% RSLogix 500 project LVD190506v3_Top.RSS, saved by version 11.00.00.00 %
PROJECT "LINCEBOT"    % processor: MicroLogix 1400 %

PROGRAM FILES
  LAD 2 "MAIN"  63 rungs  % Main Program Routine %
  LAD 8 "LOOP TIME"  6 rungs
  LAD 12 "ENABLES"  4 rungs
  LAD 14 "SPEED OUT"  3 rungs
  LAD 16 "TOTALCOUNT"  4 rungs
  LAD 19 "TESTTRIG5"  4 rungs
  LAD 20 "TESTTRIG6"  4 rungs
  LAD 21 "TESTTRIG7"  4 rungs
  LAD 22 "TESTTRIG8"  4 rungs
  LAD 24 "SKIPPED"  5 rungs
  LAD 26 "TEST TIME"  11 rungs
  LAD 70 "ALIGNFAILS"  4 rungs  % normal %
  LAD 90 "HSC TOP"  5 rungs
  LAD 100 "1 MS STI"  23 rungs  % high speed %
  LAD 103 "SPEED TOP"  8 rungs  % high speed %
  LAD 105 "P TOP"  7 rungs  % high speed %
  LAD 111 "SHIFT TOP"  15 rungs
  LAD 131 "READXFER"  3 rungs
  LAD 140 "TOP_OPTIC"  8 rungs
  LAD 141 "TOPOP_VERT"  5 rungs
  LAD 142 "TOPOP_REAL"  10 rungs
  LAD 143 "TOPOP_TEST"  13 rungs
  LAD 144 "TOP_OP_OK"  6 rungs
  LAD 150 "TOP_OPTIC"  6 rungs
  LAD 151 "TOPOP_VERT"  9 rungs
  LAD 152 "TOPOP_REAL"  11 rungs
  LAD 153 "TOPOP_TEST"  19 rungs
  LAD 154 "TOP_OP_OK"  6 rungs
  LAD 155 "OP RNG TST"  5 rungs
  LAD 190 "INS5"  21 rungs
  LAD 191 "INS5RESULT"  7 rungs
  LAD 192 "INS5PASS"  4 rungs
  LAD 193 "INS5FAIL"  3 rungs
  LAD 194 "INS5ACQ"  8 rungs
  LAD 195 "Q5TIMETEST"  5 rungs
  LAD 196 "INS5TRIG"  5 rungs
  LAD 197 "FIFO5SET"  9 rungs
  LAD 198 "FIFO5GET"  8 rungs
  LAD 199 "INSDATA5"  3 rungs
  LAD 200 "TESTFAULT5"  9 rungs
  LAD 201 "INS5FIX1"  6 rungs
  LAD 202 "INS5FIX2"  3 rungs
  LAD 204 "INS6"  21 rungs
  LAD 205 "INS6RESULT"  7 rungs
  LAD 206 "INS6PASS"  4 rungs
  LAD 207 "INS6FAIL"  3 rungs
  LAD 208 "INS6ACQ"  8 rungs
  LAD 209 "Q6TIMETEST"  5 rungs
  LAD 210 "INS6TRIG"  5 rungs
  LAD 211 "FIFO6SET"  9 rungs
  LAD 212 "FIFO6GET"  8 rungs
  LAD 213 "INSDATA6"  3 rungs
  LAD 214 "TESTFAULT6"  9 rungs
  LAD 215 "INS6FIX1"  6 rungs
  LAD 216 "INS6FIX2"  3 rungs
  LAD 218 "INS7"  21 rungs
  LAD 219 "INS7RESULT"  7 rungs
  LAD 220 "INS7PASS"  4 rungs
  LAD 221 "INS7FAIL"  3 rungs
  LAD 222 "INS7ACQ"  8 rungs
  LAD 223 "Q7TIMETEST"  5 rungs
  LAD 224 "INS7TRIG"  5 rungs
  LAD 225 "FIFO7SET"  9 rungs
  LAD 226 "FIFO7GET"  8 rungs
  LAD 227 "INSDATA7"  3 rungs
  LAD 228 "TESTFAULT7"  9 rungs
  LAD 229 "INS7FIX1"  6 rungs
  LAD 230 "INS7FIX2"  3 rungs
  LAD 232 "INS8"  21 rungs
  LAD 233 "INS8RESULT"  7 rungs
  LAD 234 "INS8PASS"  4 rungs
  LAD 235 "INS8FAIL"  3 rungs
  LAD 236 "INS8ACQ"  8 rungs
  LAD 237 "Q8TIMETEST"  5 rungs
  LAD 238 "INS8TRIG"  5 rungs
  LAD 239 "FIFO8SET"  9 rungs
  LAD 240 "FIFO8GET"  8 rungs
  LAD 241 "INSDATA8"  3 rungs
  LAD 242 "TESTFAULT8"  9 rungs
  LAD 243 "INS8FIX1"  6 rungs
  LAD 244 "INS8FIX2"  3 rungs
  LAD 249 "PASS BLOW"  25 rungs
  LAD 250 "RECERK"  10 rungs
  LAD 251 "RECERK SET"  5 rungs
  LAD 252 "RATE1"  9 rungs
  LAD 253 "RATE2"  6 rungs
  LAD 254 "RESET RATE"  6 rungs
  LAD 255 "UNUSED"  19 rungs
  LAD 149, 189, 203, 217, 231, 245: only END

DATA FILES
  O0 OUTPUT  6 elements
  I1 INPUT  8 elements
  S2 STATUS  66 elements
  B3 BINARY  64 elements
  T4 TIMER  40 elements
  C5 COUNTER  1 elements
  R6 CONTROL  20 elements
  N7 INTEGER  200 elements
  F8 FLOAT  100 elements
  B9   1 elements
  B10   1 elements
  B11   1 elements
  B12 HMI_BINARY  22 elements  % general use with hmi to avoid additional reads %
  L13  COUNTS  256 elements
  F14 HMI_FLOATS  100 elements
  N15 HMI_INTS  100 elements
  L16 HMI_LONGS  100 elements
  B17 #1 GOOD  192 elements
  B18 #2 GOOD  192 elements
  L19 I5TIMEFIFO  50 elements
  L20 I5POSFIFO  50 elements
  L21 I6TIMEFIFO  50 elements
  L22 I6POSFIFO  50 elements
  L23 I7TIMEFIFO  50 elements
  L24 I7POSFIFO  50 elements
  L25 I8TIMEFIFO  50 elements
  L26 I8POSFIFO  50 elements
  L27 RATE FIFO  50 elements
  L42 COMS  52 elements
  RI43 RI1  11 elements
  MG44 MSG1  11 elements
  B181 BLANK  256 elements  % used to wipe bs files %
  F182   50 elements
  L183   50 elements
  N184   50 elements
  B185   50 elements
  N186   50 elements
  L187   50 elements
  F188   50 elements
  B189   50 elements
  L190   50 elements
  B191   10 elements
  L192 SPD OFFSET  50 elements
  F193 SPD OFFSET  50 elements
  B194 TOP GOOD  192 elements
  B195 TOP NG  192 elements
  B196 CTRL BITS  50 elements
  N197 CTRL INTS  50 elements
  B198 TRK BITS  50 elements
  L199 TRK LONG  50 elements
  N200 TRK INTS  50 elements
  L201 INS LONG  50 elements
  B202 INS BITS  50 elements
  N203 INS INTS  50 elements
  L204 CTRL LONG  50 elements
  F205 CTRL FLTS  50 elements

LADDER 2 "MAIN"    % Main Program Routine %
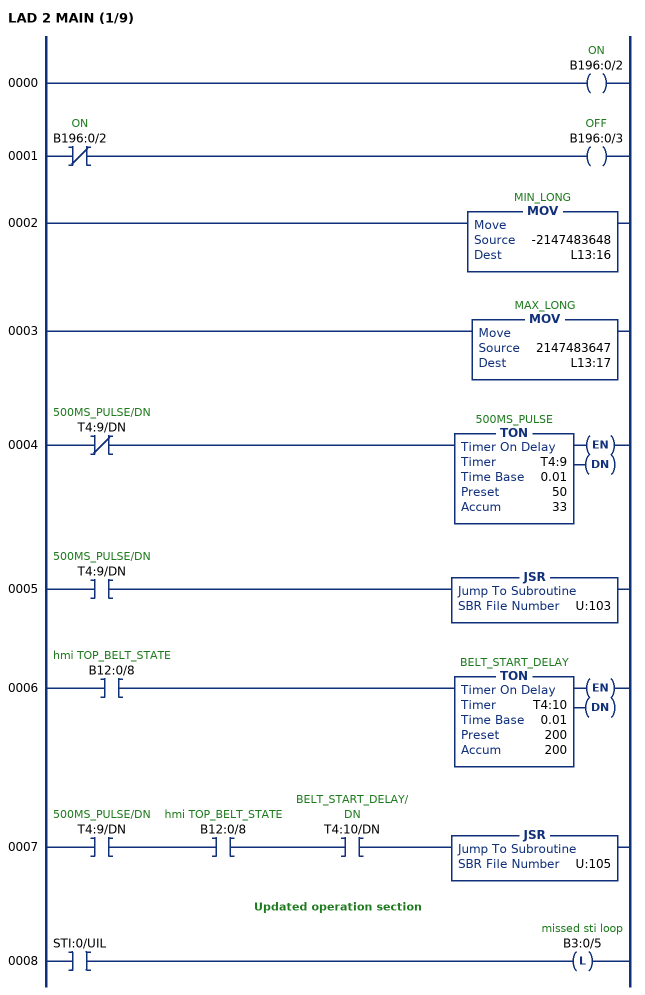
% Rung: 0 %
SOR OTE B196:0/2 EOR
%   B196:0/2  ON %
% Rung: 1 %
SOR XIO B196:0/2 OTE B196:0/3 EOR
%   B196:0/2  ON %
%   B196:0/3  OFF %
% Rung: 2 %
SOR MOV -2147483648 L13:16 EOR
%   L13:16  MIN_LONG %
% Rung: 3 %
SOR MOV 2147483647 L13:17 EOR
%   L13:17  MAX_LONG %
% Rung: 4 %
SOR XIO T4:9/DN TON T4:9 0.01 50 33 EOR
%   T4:9  500MS_PULSE %
% Rung: 5 %
SOR XIC T4:9/DN JSR U:103 EOR
%   T4:9  500MS_PULSE %
% Rung: 6 %
SOR XIC B12:0/8 TON T4:10 0.01 200 200 EOR
%   B12:0/8  TOP_BELT_STATE  "hmi" %
%   T4:10  BELT_START_DELAY %
% Rung: 7 %
SOR XIC T4:9/DN XIC B12:0/8 XIC T4:10/DN JSR U:105 EOR
%   T4:9  500MS_PULSE %
%   B12:0/8  TOP_BELT_STATE  "hmi" %
%   T4:10  BELT_START_DELAY %
% Rung: 8 %
% TITLE: Updated operation section %
SOR XIC STI:0/UIL OTL B3:0/5 EOR
%   B3:0/5  "missed sti loop" %

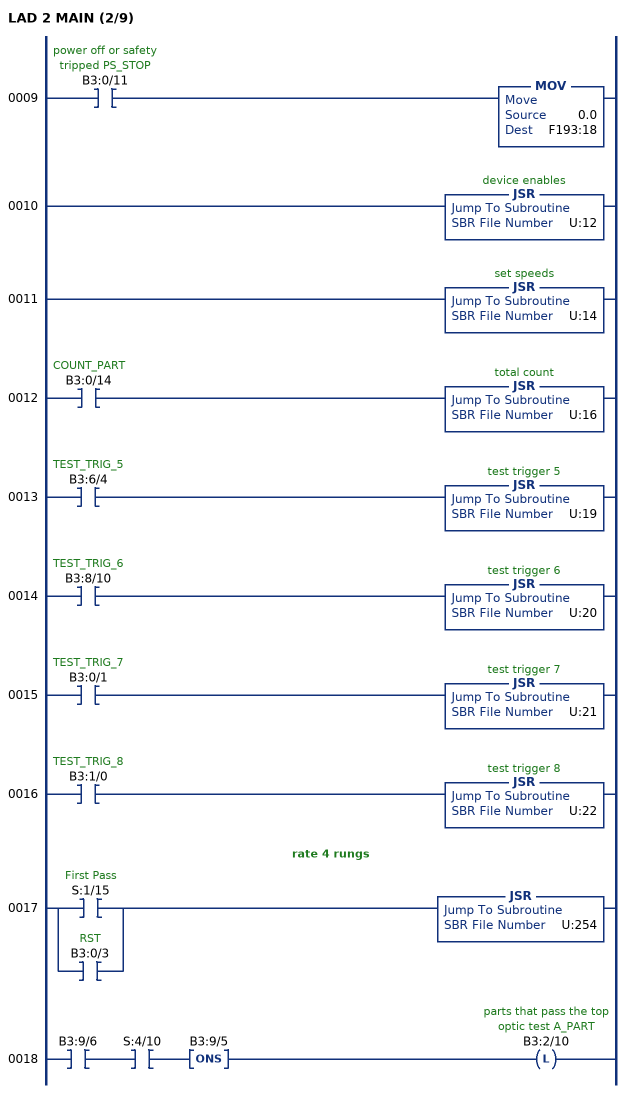
% Rung: 9 %
SOR XIC B3:0/11 MOV 0.0 F193:18 EOR
%   B3:0/11  PS_STOP  "power off or safety tripped" %
% Rung: 10 %
SOR JSR U:12 EOR
%   U:12  "device enables" %
% Rung: 11 %
SOR JSR U:14 EOR
%   U:14  "set speeds" %
% Rung: 12 %
SOR XIC B3:0/14 JSR U:16 EOR
%   B3:0/14  COUNT_PART %
%   U:16  "total count" %
% Rung: 13 %
SOR XIC B3:6/4 JSR U:19 EOR
%   B3:6/4  TEST_TRIG_5 %
%   U:19  "test trigger 5" %
% Rung: 14 %
SOR XIC B3:8/10 JSR U:20 EOR
%   B3:8/10  TEST_TRIG_6 %
%   U:20  "test trigger 6" %
% Rung: 15 %
SOR XIC B3:0/1 JSR U:21 EOR
%   B3:0/1  TEST_TRIG_7 %
%   U:21  "test trigger 7" %
% Rung: 16 %
SOR XIC B3:1/0 JSR U:22 EOR
%   B3:1/0  TEST_TRIG_8 %
%   U:22  "test trigger 8" %
% Rung: 17 %
% TITLE: rate 4 rungs %
SOR BST XIC S:1/15 NXB XIC B3:0/3 BND JSR U:254 EOR
%   S:1/15  "First Pass" %
%   B3:0/3  RST %
% Rung: 18 %
SOR XIC B3:9/6 XIC S:4/10 ONS B3:9/5 OTL B3:2/10 EOR
%   B3:2/10  A_PART  "parts that pass the top optic test" %

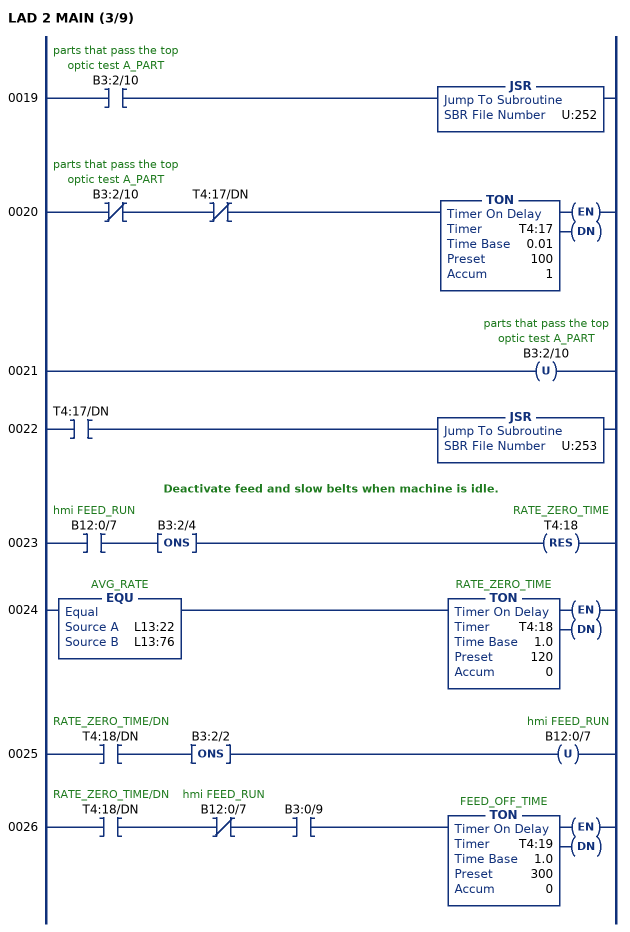
% Rung: 19 %
SOR XIC B3:2/10 JSR U:252 EOR
%   B3:2/10  A_PART  "parts that pass the top optic test" %
% Rung: 20 %
SOR XIO B3:2/10 XIO T4:17/DN TON T4:17 0.01 100 1 EOR
%   B3:2/10  A_PART  "parts that pass the top optic test" %
% Rung: 21 %
SOR OTU B3:2/10 EOR
%   B3:2/10  A_PART  "parts that pass the top optic test" %
% Rung: 22 %
SOR XIC T4:17/DN JSR U:253 EOR
% Rung: 23 %
% TITLE: Deactivate feed and slow belts when machine is idle. %
SOR XIC B12:0/7 ONS B3:2/4 RES T4:18 EOR
%   B12:0/7  FEED_RUN  "hmi" %
%   T4:18  RATE_ZERO_TIME %
% Rung: 24 %
SOR EQU L13:22 L13:76 TON T4:18 1.0 120 0 EOR
%   L13:22  AVG_RATE %
%   L13:76  PPM_AVG %
%   T4:18  RATE_ZERO_TIME %
% Rung: 25 %
SOR XIC T4:18/DN ONS B3:2/2 OTU B12:0/7 EOR
%   T4:18  RATE_ZERO_TIME %
%   B12:0/7  FEED_RUN  "hmi" %
% Rung: 26 %
SOR XIC T4:18/DN XIO B12:0/7 XIC B3:0/9 TON T4:19 1.0 300 0 EOR
%   T4:18  RATE_ZERO_TIME %
%   B12:0/7  FEED_RUN  "hmi" %
%   T4:19  FEED_OFF_TIME %

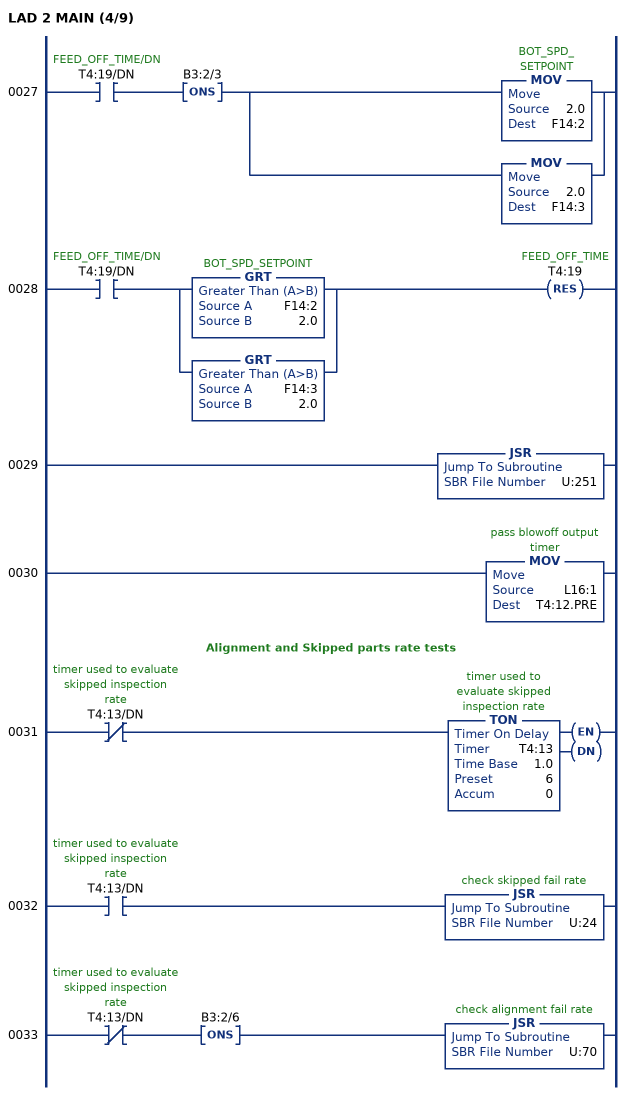
% Rung: 27 %
SOR XIC T4:19/DN ONS B3:2/3 BST MOV 2.0 F14:2 NXB MOV 2.0 F14:3 BND EOR
%   T4:19  FEED_OFF_TIME %
%   F14:2  BOT_SPD_SETPOINT %
% Rung: 28 %
SOR XIC T4:19/DN BST GRT F14:2 2.0 NXB GRT F14:3 2.0 BND RES T4:19 EOR
%   T4:19  FEED_OFF_TIME %
%   F14:2  BOT_SPD_SETPOINT %
% Rung: 29 %
SOR JSR U:251 EOR
% Rung: 30 %
SOR MOV L16:1 T4:12.PRE EOR
%   L16:1  BLOW_TIME %
%   T4:12  "pass blowoff output timer" %
% Rung: 31 %
% TITLE: Alignment and Skipped parts rate tests %
SOR XIO T4:13/DN TON T4:13 1.0 6 0 EOR
%   T4:13  "timer used to evaluate skipped inspection rate" %
% Rung: 32 %
SOR XIC T4:13/DN JSR U:24 EOR
%   T4:13  "timer used to evaluate skipped inspection rate" %
%   U:24  "check skipped fail rate" %
% Rung: 33 %
SOR XIO T4:13/DN ONS B3:2/6 JSR U:70 EOR
%   T4:13  "timer used to evaluate skipped inspection rate" %
%   U:70  "check alignment fail rate" %

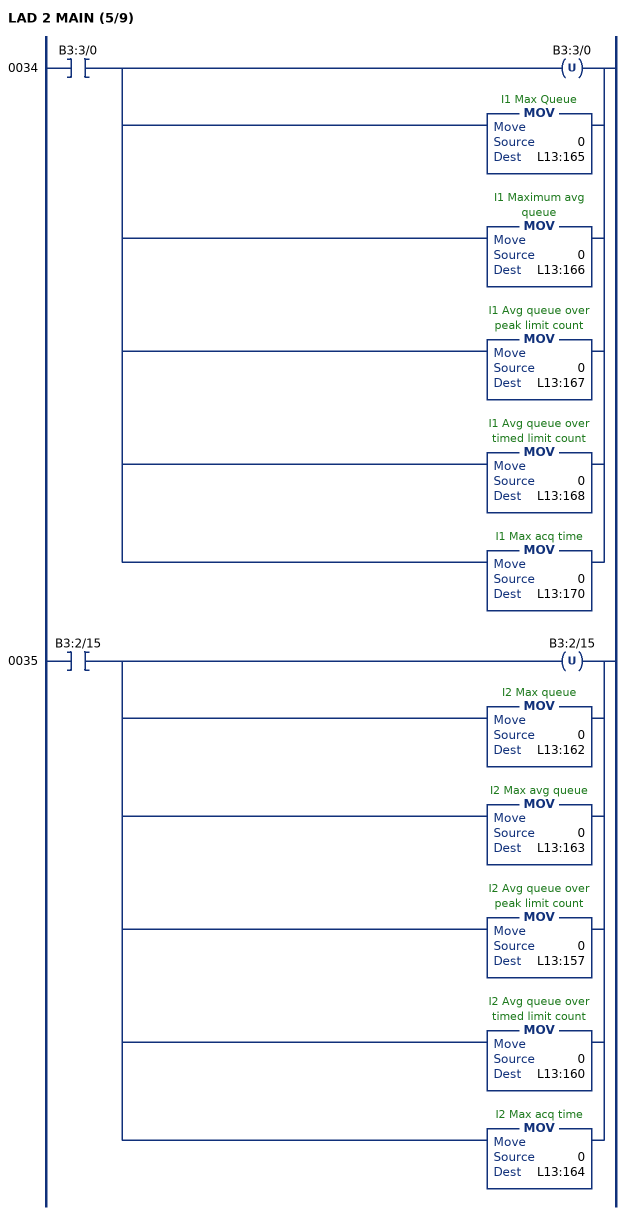
% Rung: 34 %
SOR XIC B3:3/0 BST OTU B3:3/0 NXB MOV 0 L13:165 NXB MOV 0 L13:166 NXB MOV 0 L13:167 NXB MOV 0 L13:168 NXB MOV 0 L13:170 BND EOR
%   L13:165  "I1 Max Queue" %
%   L13:166  "I1 Maximum avg queue" %
%   L13:167  "I1 Avg queue over peak limit count" %
%   L13:168  "I1 Avg queue over timed limit count" %
%   L13:170  "I1 Max acq time" %
% Rung: 35 %
SOR XIC B3:2/15 BST OTU B3:2/15 NXB MOV 0 L13:162 NXB MOV 0 L13:163 NXB MOV 0 L13:157 NXB MOV 0 L13:160 NXB MOV 0 L13:164 BND EOR
%   L13:162  "I2 Max queue" %
%   L13:163  "I2 Max avg queue" %
%   L13:157  "I2 Avg queue over peak limit count" %
%   L13:160  "I2 Avg queue over timed limit count" %
%   L13:164  "I2 Max acq time" %

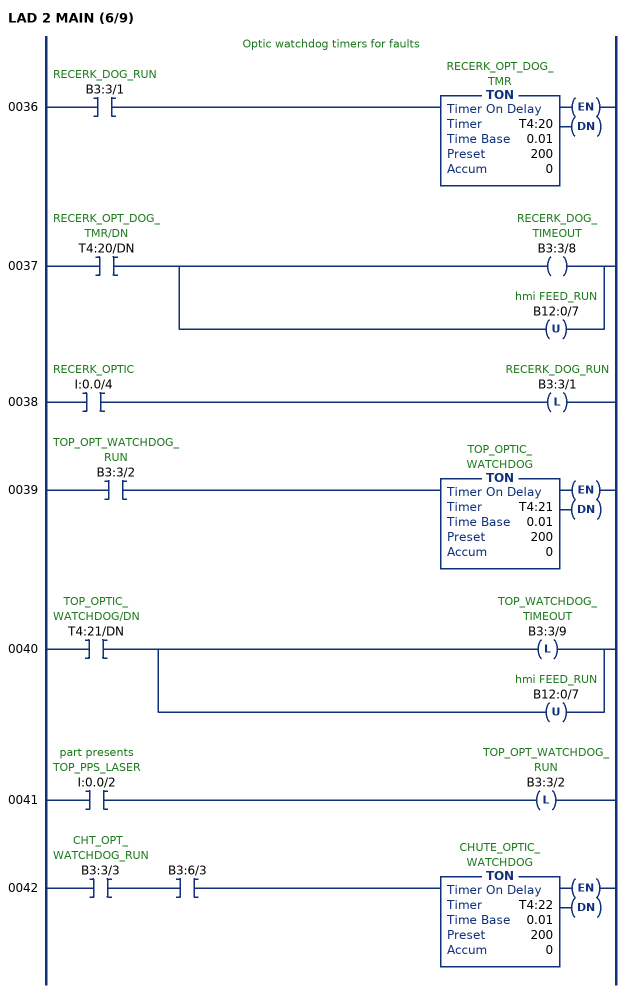
% Rung: 36 %
% Optic watchdog timers for faults %
SOR XIC B3:3/1 TON T4:20 0.01 200 0 EOR
%   B3:3/1  RECERK_DOG_RUN %
%   T4:20  RECERK_OPT_DOG_TMR %
% Rung: 37 %
SOR XIC T4:20/DN BST OTE B3:3/8 NXB OTU B12:0/7 BND EOR
%   T4:20  RECERK_OPT_DOG_TMR %
%   B3:3/8  RECERK_DOG_TIMEOUT %
%   B12:0/7  FEED_RUN  "hmi" %
% Rung: 38 %
SOR XIC I:0.0/4 OTL B3:3/1 EOR
%   I:0.0/4  RECERK_OPTIC %
%   B3:3/1  RECERK_DOG_RUN %
% Rung: 39 %
SOR XIC B3:3/2 TON T4:21 0.01 200 0 EOR
%   B3:3/2  TOP_OPT_WATCHDOG_RUN %
%   T4:21  TOP_OPTIC_WATCHDOG %
% Rung: 40 %
SOR XIC T4:21/DN BST OTL B3:3/9 NXB OTU B12:0/7 BND EOR
%   T4:21  TOP_OPTIC_WATCHDOG %
%   B3:3/9  TOP_WATCHDOG_TIMEOUT %
%   B12:0/7  FEED_RUN  "hmi" %
% Rung: 41 %
SOR XIC I:0.0/2 OTL B3:3/2 EOR
%   I:0.0/2  TOP_PPS_LASER  "part presents" %
%   B3:3/2  TOP_OPT_WATCHDOG_RUN %
% Rung: 42 %
SOR XIC B3:3/3 XIC B3:6/3 TON T4:22 0.01 200 0 EOR
%   B3:3/3  CHT_OPT_WATCHDOG_RUN %
%   T4:22  CHUTE_OPTIC_WATCHDOG %

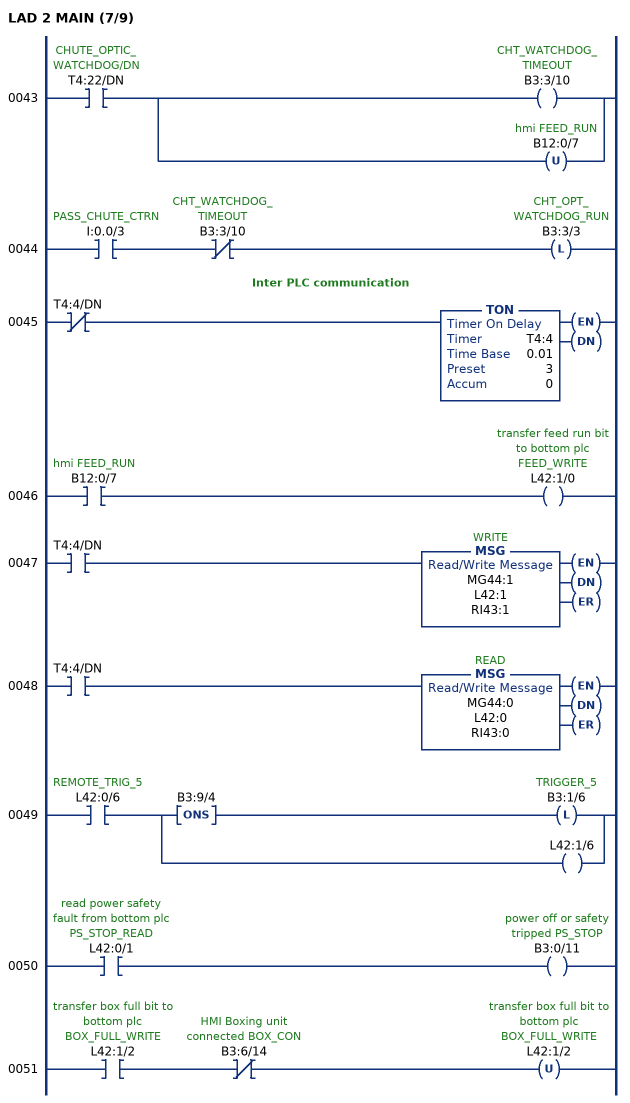
% Rung: 43 %
SOR XIC T4:22/DN BST OTE B3:3/10 NXB OTU B12:0/7 BND EOR
%   T4:22  CHUTE_OPTIC_WATCHDOG %
%   B3:3/10  CHT_WATCHDOG_TIMEOUT %
%   B12:0/7  FEED_RUN  "hmi" %
% Rung: 44 %
SOR XIC I:0.0/3 XIO B3:3/10 OTL B3:3/3 EOR
%   I:0.0/3  PASS_CHUTE_CTRN %
%   B3:3/10  CHT_WATCHDOG_TIMEOUT %
%   B3:3/3  CHT_OPT_WATCHDOG_RUN %
% Rung: 45 %
% TITLE: Inter PLC communication %
SOR XIO T4:4/DN TON T4:4 0.01 3 0 EOR
% Rung: 46 %
SOR XIC B12:0/7 OTE L42:1/0 EOR
%   B12:0/7  FEED_RUN  "hmi" %
%   L42:1/0  FEED_WRITE  "transfer feed run bit to bottom plc" %
% Rung: 47 %
SOR XIC T4:4/DN MSG MG44:1 L42:1 RI43:1 EOR
%   MSG set-up: 500CPU Write | 33 | 1 | L42:0 | L42:1 | 0 | 0 | 0 | 192.168.222.100:0 | 0 | 0 | 192.168.222.100 | RI43:1 %
%   MG44:1  WRITE %
%   L42:1  WRITE_BITS %
% Rung: 48 %
SOR XIC T4:4/DN MSG MG44:0 L42:0 RI43:0 EOR
%   MSG set-up: 500CPU Read | 33 | 1 | L42:1 | L42:0 | 0 | 0 | 0 | 192.168.222.100:0 | 0 | 0 | 192.168.222.100 | RI43:0 %
%   MG44:0  READ %
%   L42:0  READ_BITS %
% Rung: 49 %
SOR XIC L42:0/6 BST ONS B3:9/4 OTL B3:1/6 NXB OTE L42:1/6 BND EOR
%   L42:0/6  REMOTE_TRIG_5 %
%   B3:1/6  TRIGGER_5 %
% Rung: 50 %
SOR XIC L42:0/1 OTE B3:0/11 EOR
%   L42:0/1  PS_STOP_READ  "read power safety fault from bottom plc" %
%   B3:0/11  PS_STOP  "power off or safety tripped" %
% Rung: 51 %
SOR XIC L42:1/2 XIO B3:6/14 OTU L42:1/2 EOR
%   L42:1/2  BOX_FULL_WRITE  "transfer box full bit to bottom plc" %
%   B3:6/14  BOX_CON  "HMI Boxing unit connected" %

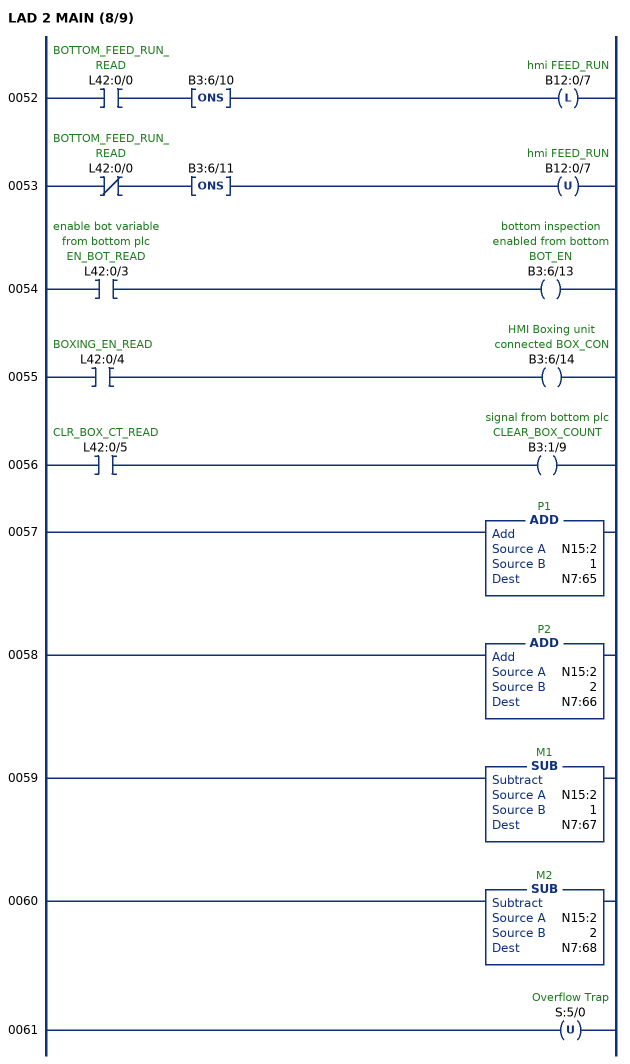
% Rung: 52 %
SOR XIC L42:0/0 ONS B3:6/10 OTL B12:0/7 EOR
%   L42:0/0  BOTTOM_FEED_RUN_READ %
%   B12:0/7  FEED_RUN  "hmi" %
% Rung: 53 %
SOR XIO L42:0/0 ONS B3:6/11 OTU B12:0/7 EOR
%   L42:0/0  BOTTOM_FEED_RUN_READ %
%   B12:0/7  FEED_RUN  "hmi" %
% Rung: 54 %
SOR XIC L42:0/3 OTE B3:6/13 EOR
%   L42:0/3  EN_BOT_READ  "enable bot variable from bottom plc" %
%   B3:6/13  BOT_EN  "bottom inspection enabled from bottom" %
% Rung: 55 %
SOR XIC L42:0/4 OTE B3:6/14 EOR
%   L42:0/4  BOXING_EN_READ %
%   B3:6/14  BOX_CON  "HMI Boxing unit connected" %
% Rung: 56 %
SOR XIC L42:0/5 OTE B3:1/9 EOR
%   L42:0/5  CLR_BOX_CT_READ %
%   B3:1/9  CLEAR_BOX_COUNT  "signal from bottom plc" %
% Rung: 57 %
SOR ADD N15:2 1 N7:65 EOR
%   N15:2  BLOW_PT %
%   N7:65  P1 %
% Rung: 58 %
SOR ADD N15:2 2 N7:66 EOR
%   N15:2  BLOW_PT %
%   N7:66  P2 %
% Rung: 59 %
SOR SUB N15:2 1 N7:67 EOR
%   N15:2  BLOW_PT %
%   N7:67  M1 %
% Rung: 60 %
SOR SUB N15:2 2 N7:68 EOR
%   N15:2  BLOW_PT %
%   N7:68  M2 %
% Rung: 61 %
SOR OTU S:5/0 EOR
%   S:5/0  "Overflow Trap" %

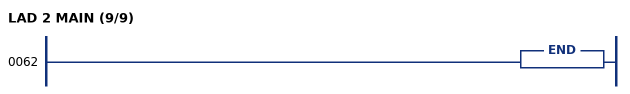
% Rung: 62 %
SOR END EOR

LADDER 8 "LOOP TIME"
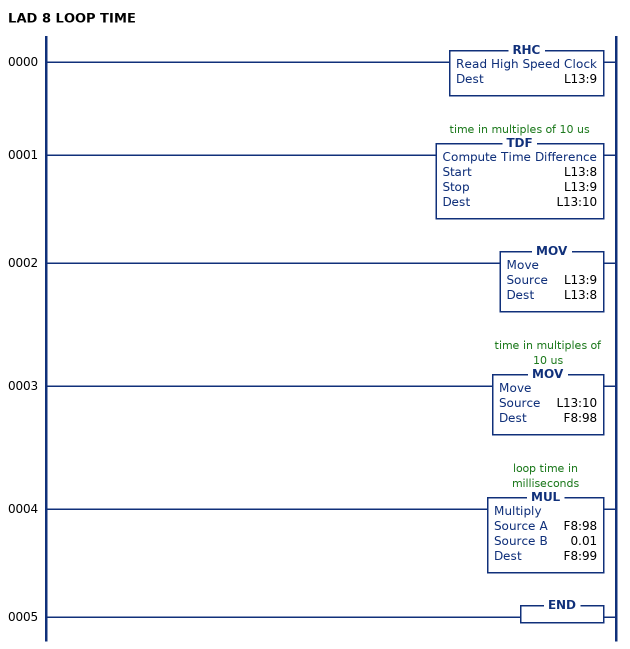
% Rung: 0 %
SOR RHC L13:9 EOR
% Rung: 1 %
SOR TDF L13:8 L13:9 L13:10 EOR
%   L13:10  "time in multiples of 10 us" %
% Rung: 2 %
SOR MOV L13:9 L13:8 EOR
% Rung: 3 %
SOR MOV L13:10 F8:98 EOR
%   L13:10  "time in multiples of 10 us" %
%   F8:98  "time in multiples of 10 us" %
% Rung: 4 %
SOR MUL F8:98 0.01 F8:99 EOR
%   F8:98  "time in multiples of 10 us" %
%   F8:99  "loop time in milliseconds" %
% Rung: 5 %
SOR END EOR

LADDER 12 "ENABLES"
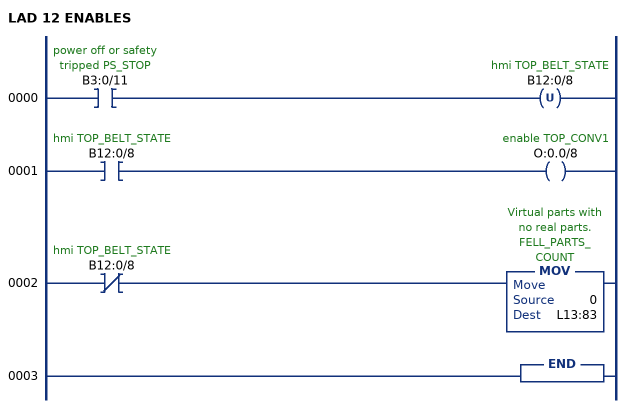
% Rung: 0 %
SOR XIC B3:0/11 OTU B12:0/8 EOR
%   B3:0/11  PS_STOP  "power off or safety tripped" %
%   B12:0/8  TOP_BELT_STATE  "hmi" %
% Rung: 1 %
SOR XIC B12:0/8 OTE O:0.0/8 EOR
%   B12:0/8  TOP_BELT_STATE  "hmi" %
%   O:0.0/8  TOP_CONV1  "enable" %
% Rung: 2 %
SOR XIO B12:0/8 MOV 0 L13:83 EOR
%   B12:0/8  TOP_BELT_STATE  "hmi" %
%   L13:83  FELL_PARTS_COUNT  "Virtual parts with no real parts." %
% Rung: 3 %
SOR END EOR

LADDER 14 "SPEED OUT"
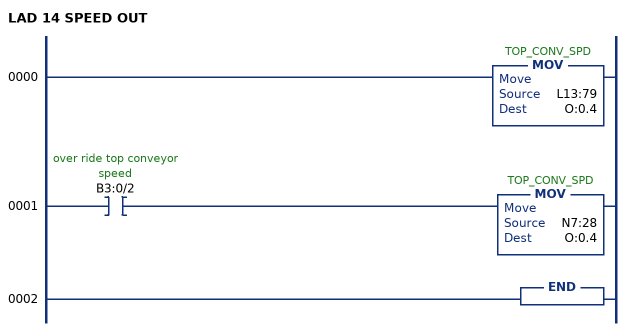
% Rung: 0 %
SOR MOV L13:79 O:0.4 EOR
%   L13:79  SCALED_TOP_VALUE %
%   O:0.4  TOP_CONV_SPD %
% Rung: 1 %
SOR XIC B3:0/2 MOV N7:28 O:0.4 EOR
%   B3:0/2  "over ride top conveyor speed" %
%   O:0.4  TOP_CONV_SPD %
% Rung: 2 %
SOR END EOR

LADDER 16 "TOTALCOUNT"
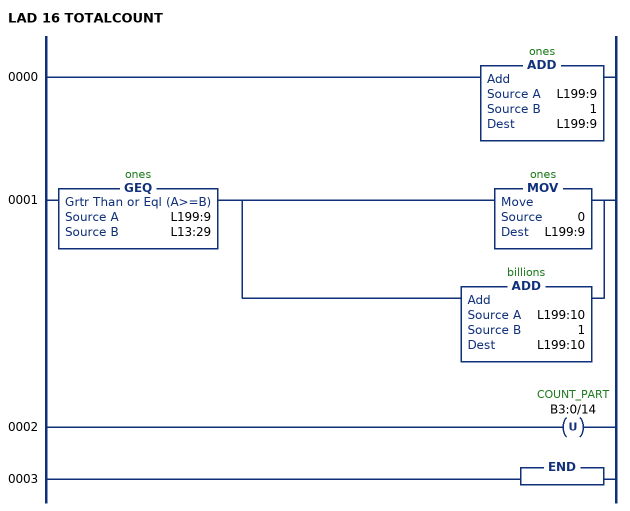
% Rung: 0 %
SOR ADD L199:9 1 L199:9 EOR
%   L199:9  "ones" %
% Rung: 1 %
SOR GEQ L199:9 L13:29 BST MOV 0 L199:9 NXB ADD L199:10 1 L199:10 BND EOR
%   L199:9  "ones" %
%   L13:29  "maximum of the longest acquire time allowed if maximum acquire time fault is enabled" %
%   L199:10  "billions" %
% Rung: 2 %
SOR OTU B3:0/14 EOR
%   B3:0/14  COUNT_PART %
% Rung: 3 %
SOR END EOR

LADDER 19 "TESTTRIG5"
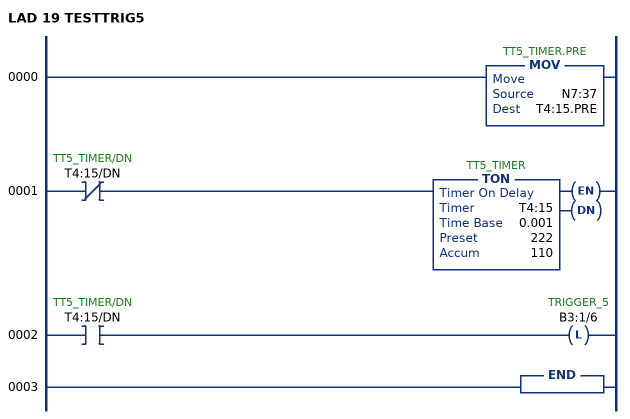
% Rung: 0 %
SOR MOV N7:37 T4:15.PRE EOR
%   T4:15  TT5_TIMER %
% Rung: 1 %
SOR XIO T4:15/DN TON T4:15 0.001 222 110 EOR
%   T4:15  TT5_TIMER %
% Rung: 2 %
SOR XIC T4:15/DN OTL B3:1/6 EOR
%   T4:15  TT5_TIMER %
%   B3:1/6  TRIGGER_5 %
% Rung: 3 %
SOR END EOR

LADDER 20 "TESTTRIG6"
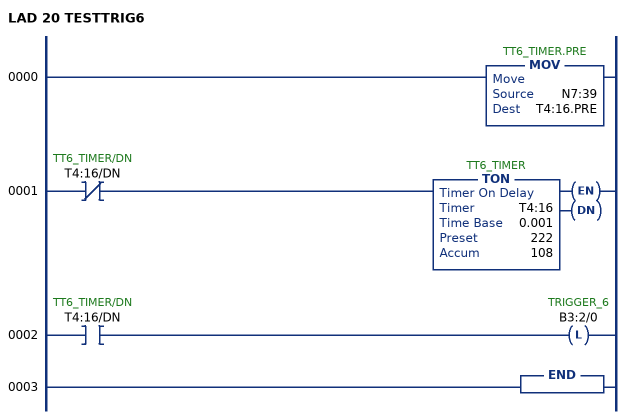
% Rung: 0 %
SOR MOV N7:39 T4:16.PRE EOR
%   T4:16  TT6_TIMER %
% Rung: 1 %
SOR XIO T4:16/DN TON T4:16 0.001 222 108 EOR
%   T4:16  TT6_TIMER %
% Rung: 2 %
SOR XIC T4:16/DN OTL B3:2/0 EOR
%   T4:16  TT6_TIMER %
%   B3:2/0  TRIGGER_6 %
% Rung: 3 %
SOR END EOR

LADDER 21 "TESTTRIG7"
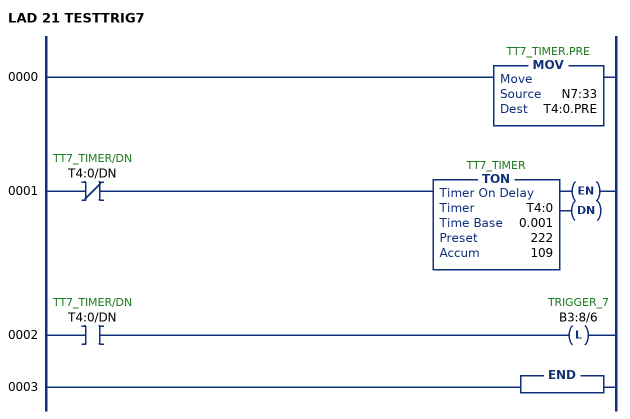
% Rung: 0 %
SOR MOV N7:33 T4:0.PRE EOR
%   T4:0  TT7_TIMER %
% Rung: 1 %
SOR XIO T4:0/DN TON T4:0 0.001 222 109 EOR
%   T4:0  TT7_TIMER %
% Rung: 2 %
SOR XIC T4:0/DN OTL B3:8/6 EOR
%   T4:0  TT7_TIMER %
%   B3:8/6  TRIGGER_7 %
% Rung: 3 %
SOR END EOR

LADDER 22 "TESTTRIG8"
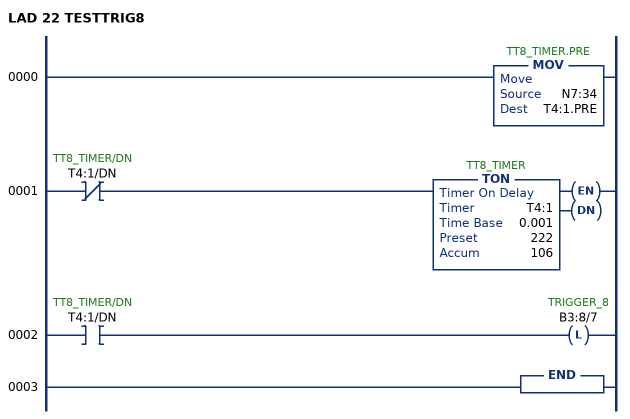
% Rung: 0 %
SOR MOV N7:34 T4:1.PRE EOR
%   T4:1  TT8_TIMER %
% Rung: 1 %
SOR XIO T4:1/DN TON T4:1 0.001 222 106 EOR
%   T4:1  TT8_TIMER %
% Rung: 2 %
SOR XIC T4:1/DN OTL B3:8/7 EOR
%   T4:1  TT8_TIMER %
%   B3:8/7  TRIGGER_8 %
% Rung: 3 %
SOR END EOR

LADDER 24 "SKIPPED"
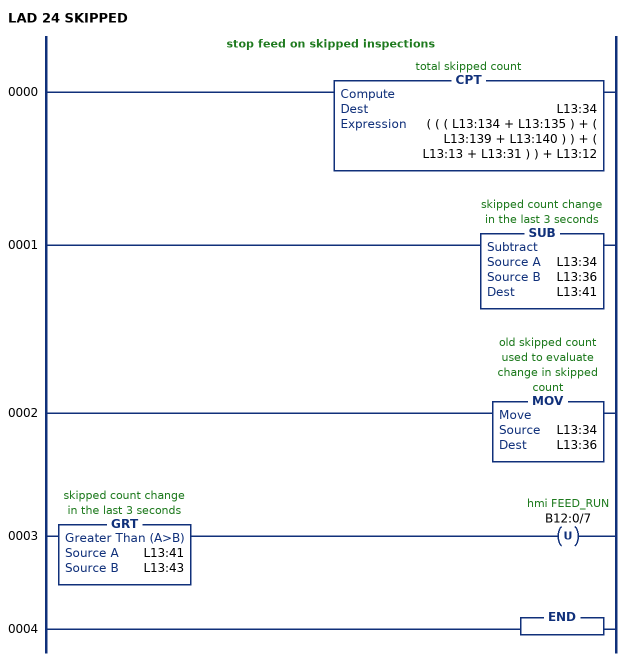
% Rung: 0 %
% TITLE: stop feed on skipped inspections %
SOR CPT L13:34 " ( ( ( L13:134 + L13:135 ) + ( L13:139 + L13:140 ) ) + ( L13:13 + L13:31 ) ) + L13:12 " EOR
%   L13:34  "total skipped count" %
%   L13:134  "too wide bottom" %
%   L13:135  "too close bottom" %
%   L13:139  "too close top count" %
%   L13:140  "too wide top count" %
%   L13:13  SKIP1  "skipped 1 count" %
%   L13:31  SKIP5  "skipped 5 count" %
%   L13:12  SKIP6  "skipped 6 count" %
% Rung: 1 %
SOR SUB L13:34 L13:36 L13:41 EOR
%   L13:34  "total skipped count" %
%   L13:36  "old skipped count used to evaluate change in skipped count" %
%   L13:41  "skipped count change in the last 3 seconds" %
% Rung: 2 %
SOR MOV L13:34 L13:36 EOR
%   L13:34  "total skipped count" %
%   L13:36  "old skipped count used to evaluate change in skipped count" %
% Rung: 3 %
SOR GRT L13:41 L13:43 OTU B12:0/7 EOR
%   L13:41  "skipped count change in the last 3 seconds" %
%   L13:43  "trigger count 1" %
%   B12:0/7  FEED_RUN  "hmi" %
% Rung: 4 %
SOR END EOR

LADDER 26 "TEST TIME"
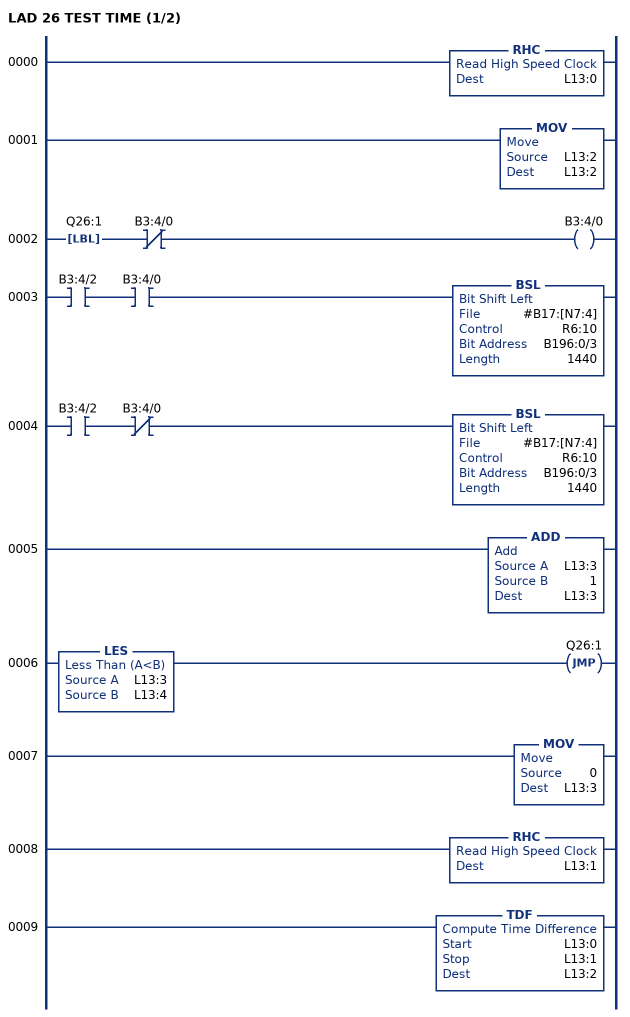
% Rung: 0 %
SOR RHC L13:0 EOR
% Rung: 1 %
SOR MOV L13:2 L13:2 EOR
% Rung: 2 %
SOR LBL Q26:1 XIO B3:4/0 OTE B3:4/0 EOR
% Rung: 3 %
SOR XIC B3:4/2 XIC B3:4/0 BSL #B17:[N7:4] R6:10 B196:0/3 1440 EOR
%   B196:0/3  OFF %
% Rung: 4 %
SOR XIC B3:4/2 XIO B3:4/0 BSL #B17:[N7:4] R6:10 B196:0/3 1440 EOR
%   B196:0/3  OFF %
% Rung: 5 %
SOR ADD L13:3 1 L13:3 EOR
% Rung: 6 %
SOR LES L13:3 L13:4 JMP Q26:1 EOR
% Rung: 7 %
SOR MOV 0 L13:3 EOR
% Rung: 8 %
SOR RHC L13:1 EOR
% Rung: 9 %
SOR TDF L13:0 L13:1 L13:2 EOR

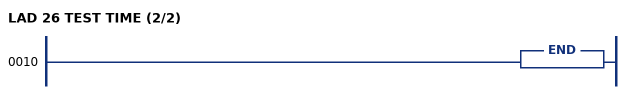
% Rung: 10 %
SOR END EOR

LADDER 70 "ALIGNFAILS"    % normal %
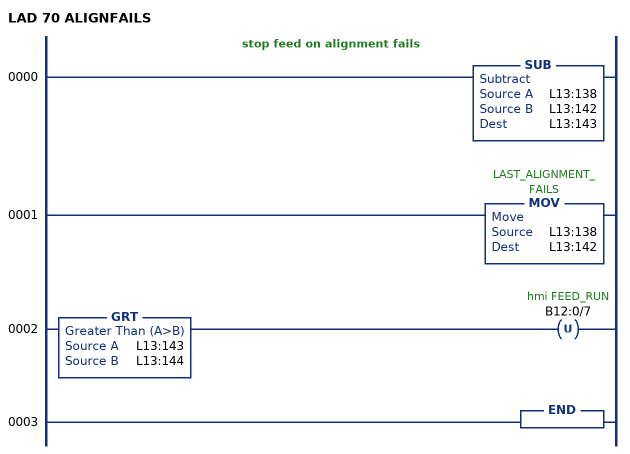
% Rung: 0 %
% TITLE: stop feed on alignment fails %
SOR SUB L13:138 L13:142 L13:143 EOR
%   L13:138  "alignment fail counts" %
%   L13:142  LAST_ALIGNMENT_FAILS %
% Rung: 1 %
SOR MOV L13:138 L13:142 EOR
%   L13:138  "alignment fail counts" %
%   L13:142  LAST_ALIGNMENT_FAILS %
% Rung: 2 %
SOR GRT L13:143 L13:144 OTU B12:0/7 EOR
%   B12:0/7  FEED_RUN  "hmi" %
% Rung: 3 %
SOR END EOR

LADDER 90 "HSC TOP"
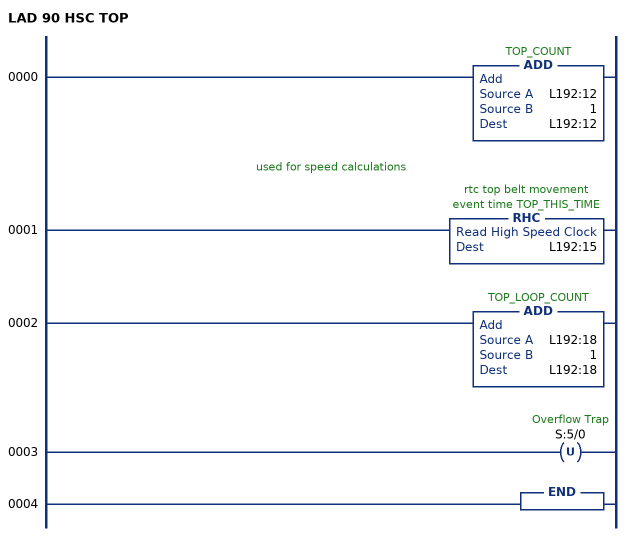
% Rung: 0 %
SOR ADD L192:12 1 L192:12 EOR
%   L192:12  TOP_COUNT %
% Rung: 1 %
% used for speed calculations %
SOR RHC L192:15 EOR
%   L192:15  TOP_THIS_TIME  "rtc top belt movement event time" %
% Rung: 2 %
SOR ADD L192:18 1 L192:18 EOR
%   L192:18  TOP_LOOP_COUNT %
% Rung: 3 %
SOR OTU S:5/0 EOR
%   S:5/0  "Overflow Trap" %
% Rung: 4 %
SOR END EOR

LADDER 100 "1 MS STI"    % high speed %
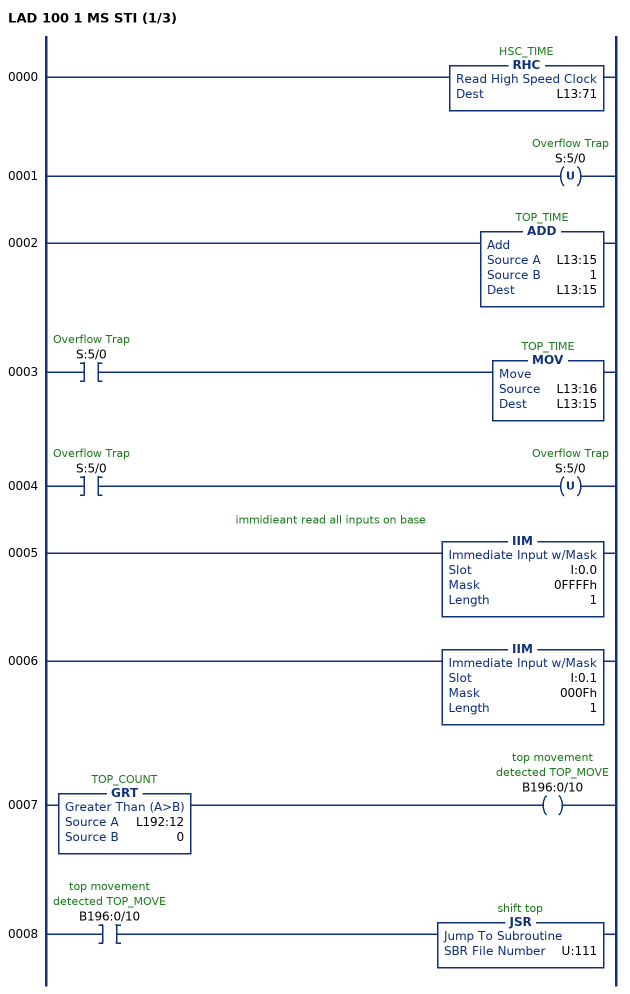
% Rung: 0 %
SOR RHC L13:71 EOR
%   L13:71  HSC_TIME %
% Rung: 1 %
SOR OTU S:5/0 EOR
%   S:5/0  "Overflow Trap" %
% Rung: 2 %
SOR ADD L13:15 1 L13:15 EOR
%   L13:15  TOP_TIME %
% Rung: 3 %
SOR XIC S:5/0 MOV L13:16 L13:15 EOR
%   S:5/0  "Overflow Trap" %
%   L13:16  MIN_LONG %
%   L13:15  TOP_TIME %
% Rung: 4 %
SOR XIC S:5/0 OTU S:5/0 EOR
%   S:5/0  "Overflow Trap" %
% Rung: 5 %
% immidieant read all inputs on base %
SOR IIM I:0.0 0FFFFh 1 EOR
% Rung: 6 %
SOR IIM I:0.1 000Fh 1 EOR
% Rung: 7 %
SOR GRT L192:12 0 OTE B196:0/10 EOR
%   L192:12  TOP_COUNT %
%   B196:0/10  TOP_MOVE  "top movement detected" %
% Rung: 8 %
SOR XIC B196:0/10 JSR U:111 EOR
%   B196:0/10  TOP_MOVE  "top movement detected" %
%   U:111  "shift top" %

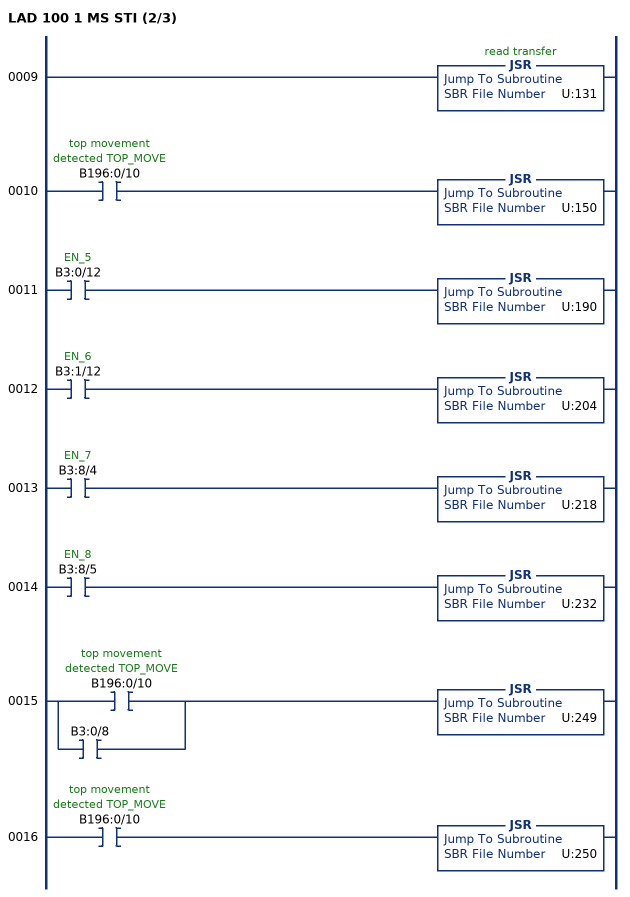
% Rung: 9 %
SOR JSR U:131 EOR
%   U:131  "read transfer" %
% Rung: 10 %
SOR XIC B196:0/10 JSR U:150 EOR
%   B196:0/10  TOP_MOVE  "top movement detected" %
% Rung: 11 %
SOR XIC B3:0/12 JSR U:190 EOR
%   B3:0/12  EN_5 %
% Rung: 12 %
SOR XIC B3:1/12 JSR U:204 EOR
%   B3:1/12  EN_6 %
% Rung: 13 %
SOR XIC B3:8/4 JSR U:218 EOR
%   B3:8/4  EN_7 %
% Rung: 14 %
SOR XIC B3:8/5 JSR U:232 EOR
%   B3:8/5  EN_8 %
% Rung: 15 %
SOR BST XIC B196:0/10 NXB XIC B3:0/8 BND JSR U:249 EOR
%   B196:0/10  TOP_MOVE  "top movement detected" %
% Rung: 16 %
SOR XIC B196:0/10 JSR U:250 EOR
%   B196:0/10  TOP_MOVE  "top movement detected" %

